FUNCTION_BLOCK FB_AlarmManager
VAR_INPUT
END_VAR
VAR_OUTPUT
END_VAR
VAR
END_VAR

END_FUNCTION_BLOCK

(* stored: Version 1.1.0.1, ProductVersion 3.1.4026.18
   POU FB_AlarmManager: Id {f6bca294-1f03-41a5-bfcd-6e3752b44b89}, SpecialFunc None *)
